// Mitsubishi GX Works2 project: KemNghiaDrillV1.5   PLC: FX3U/FX3UC

// global labels: Global1
VAR_GLOBAL
  XXLimitN AT M8344 : BOOL;
  XXLimitP AT M8343 : BOOL;
  XXBusy AT M8340 : BOOL;
  XXInterruptInverse AT M8347 : BOOL;
  XXPos AT D8340 : DINT;
  XXAccelTime AT D8348 : INT;
  XXDecelTime AT D8349 : INT;
  XXPosView AT D0 : DINT;
  XXTarPos AT D2 : DINT;
  XXFeed AT D4 : DINT;
  XXTarR AT M0 : BOOL;
  XXTarRSkip AT D6 : INT;
  XXManualN AT M1 : BOOL;
  XXManualP AT M2 : BOOL;
  XXOn AT M3 : BOOL;
  XXRun AT M4 : BOOL;
  XXDirection AT M5 : BOOL;
  XXMinI AT X000 : BOOL;
  XXAlarmI AT X004 : BOOL;
  XXReadyI AT X010 : BOOL;
  XXPulseO AT Y000 : BOOL;
  XXDirectionO AT Y004 : BOOL;
  XXOnO AT Y002 : BOOL;
  MachineReady AT M6 : BOOL;
  MachineReadyTimer AT TC0 : BOOL;
  Run AT M7 : BOOL;
  RunI AT X001 : BOOL;
  RunStop AT M8 : BOOL;
  RunStopI AT X002 : BOOL;
  RunStart AT M9 : BOOL;
  RunAuto AT M10 : BOOL;
  RunAutoEnableTimer AT TC1 : BOOL;
  RunTest AT M11 : BOOL;
  RunTestMeasureTimer AT TC246 : BOOL;
  RunTestMeasureTimerValue AT TN246 : INT;
  PositionArray AT D1000 : ARRAY [0..7] OF DINT;
  RunState AT D7 : INT;
  RunStateNext AT M12 : BOOL;
  RunStateDisc AT D8 : INT;
  RunStateDiscNext AT M13 : BOOL;
  RunStateFoilExtract AT D9 : INT;
  RunStateFoilExtractNext AT M14 : BOOL;
  RunStateDrill AT D10 : INT;
  RunStateDrillNext AT M15 : BOOL;
  RunStateFoilOut AT D11 : INT;
  RunStateFoilOutNext AT M16 : BOOL;
  DiscDRVIOffset AT D12 : DINT;
  DiscDRVIOffsetBefore AT D14 : DINT;
  DiscDRVIFrequency AT D16 : DINT;
  DiscSectorCount AT D18 : INT;
  DiscStepCount AT D19 : INT;
  DiscTest AT M17 : BOOL;
  DiscTestDelayTimer AT TC2 : BOOL;
  DiscTestMeasureTimer AT TC247 : BOOL;
  DiscTestMeasureTimerValue AT TN247 : INT;
  FoilExtractTopN AT M18 : BOOL;
  FoilExtractTopNTimer AT TC3 : BOOL;
  FoilExtractTopP AT M19 : BOOL;
  FoilExtractTopPTimer AT TC4 : BOOL;
  FoilExtractTopNI AT X003 : BOOL;
  FoilExtractTopPI AT X005 : BOOL;
  FoilExtractTop AT M20 : BOOL;
  FoilExtractTopO AT Y001 : BOOL;
  FoilExtractTopBackDelay AT D20 : INT;
  FoilExtractBotN AT M21 : BOOL;
  FoilExtractBotNTimer AT TC5 : BOOL;
  FoilExtractBotP AT M22 : BOOL;
  FoilExtractBotPTimer AT TC6 : BOOL;
  FoilExtractBotNI AT X006 : BOOL;
  FoilExtractBotPI AT X007 : BOOL;
  FoilExtractBot AT M23 : BOOL;
  FoilExtractBotO AT Y003 : BOOL;
  FoilExtractBotBackDelay AT D21 : INT;
  FoilExtractTimer AT TC7 : BOOL;
  Drill AT M24 : BOOL;
  DrillO AT Y005 : BOOL;
  DrillHold AT M25 : BOOL;
  DrillHoldO AT Y006 : BOOL;
  DrillN AT M26 : BOOL;
  DrillP AT M27 : BOOL;
  DrillNI AT X011 : BOOL;
  DrillPI AT X012 : BOOL;
  DrillIgnore AT M28 : BOOL;
  DrillIgnoreEnableTimer AT TC8 : BOOL;
  DrillIgnoreDisableTimer AT TC9 : BOOL;
  DrillIgnoreO AT Y017 : BOOL;
  DrillTimer AT TC10 : BOOL;
  FoilOutN AT M29 : BOOL;
  FoilOutNTimer AT TC11 : BOOL;
  FoilOutP AT M30 : BOOL;
  FoilOutPTimer AT TC12 : BOOL;
  FoilOutNI AT X013 : BOOL;
  FoilOutPI AT X014 : BOOL;
  FoilOut AT M31 : BOOL;
  FoilOutO AT Y007 : BOOL;
  AirBurst AT M32 : BOOL;
  AirBurstO AT Y010 : BOOL;
  AirBurstTimer AT TC13 : BOOL;
END_VAR

// task Task_01 (event TRUE, interval 0, priority 31): POU_01

PROGRAM POU_01
VAR
  fTmp : BOOL;
END_VAR
SET(M8002, M8336);
MOV(M8002, HFFF0, D8336);
RST(M8002, XXInterruptInverse);
ZRST(M8002, RunState, RunStateFoilOut);
MOV(M8002, 250, XXAccelTime);
MOV(M8002, 250, XXDecelTime);
SET(M8002, FoilExtractTop);
SET(M8002, FoilExtractBot);
RST(M8002, Drill);
MOV(M8002, 10, FoilExtractTopBackDelay);
MOV(M8002, 10, FoilExtractBotBackDelay);
RST(M8002, DiscTest);

MOV(M8002, 8, DiscSectorCount);
DMOV(M8002, 8704, XXFeed);
DMOV(M8002, 4096, PositionArray[0]);
DMOV(M8002, 4096 * 1, PositionArray[1]);
DMOV(M8002, 4096 * 2, PositionArray[2]);
DMOV(M8002, 4096 * 3, PositionArray[3]);
DMOV(M8002, 4096 * 4, PositionArray[4]);
DMOV(M8002, 4096 * 5, PositionArray[5]);
DMOV(M8002, 4096 * 6, PositionArray[6]);
DMOV(M8002, 4096 * 7, PositionArray[7]);

OUT_T(M8000 AND NOT MachineReady, MachineReadyTimer, 10);
SET(MachineReadyTimer, MachineReady);

DMOV(M8002, 128, DiscDRVIOffset);
DMOV(M8002, 256, DiscDRVIOffsetBefore); (*offset beforce must larger than offset*)
DMOV(M8002, 512, DiscDRVIFrequency);

SET(MachineReady AND Run AND RunState = 0, fTmp);
RST(fTmp, Run);
MOV(fTmp, 1, RunState);
RST(fTmp, fTmp);
SET(RunStop, fTmp);
RST(fTmp, RunStop);
ZRST(fTmp, RunState, RunStateFoilOut);
ZRST(fTmp, RunStateNext, RunStateFoilOutNext);
RST(fTmp, XXRun);
RST(fTmp, XXOn);
RST(fTmp, FoilOut);
RST(fTmp, fTmp);

INC(RunStateNext, RunState);
INC(RunStateDiscNext, RunStateDisc);
INC(RunStateFoilExtractNext, RunStateFoilExtract);
INC(RunStateDrillNext, RunStateDrill);
INC(RunStateFoilOutNext, RunStateFoilOut);
ZRST(M8000, RunStateNext, RunStateFoilOutNext);
DECO(M8000, RunState, 6, M100); 
DECO(M8000, RunStateDisc, 6, M200); DECO(M8000, RunStateDisc, 6, M1200); ZRST(NOT (XXTarR AND XXReadyI AND NOT XXAlarmI), M1200, M1263);
DECO(M8000, RunStateFoilExtract, 6, M300);
DECO(M8000, RunStateDrill, 6, M400);
DECO(M8000, RunStateFoilOut, 6, M500);

(*||||||||||Main*)
(*start run, start disc get origin*)
SET(M101, RunStart);
SET(M101, RunStateNext);
MOV(M101, 1, RunStateDisc);
(*wait disc get origin done, move to wait run command*)
MOV(M102 AND M1260, 11, RunState);
(*wait run command*)
SET(M111 AND RunAuto, fTmp);
SET(M111 AND NOT RunAuto AND Run, fTmp);
RST(fTmp, Run);
MOV(fTmp AND NOT RunStart, 21, RunStateDisc);
RST(fTmp AND RunStart, RunStart);
SET(fTmp, RunStateNext);
RST(fTmp, fTmp);
(*got run command*)
SET(M112, RunStateNext);
(*wait disc move to next position*)
SET(M113 AND M1260, RunStateNext);
(*start cycle*)
MOV(M114, 1, RunStateFoilExtract);
MOV(M114, 1, RunStateDrill);
MOV(M114, 1, RunStateFoilOut);
SET(M114, RunStateNext);
(*wait all completed, back to wait run command*)
MOV(M115 AND M1260 AND M360 AND M460 AND M560, 11, RunState);
(*test*)
RST(RunTest AND M112, RunTestMeasureTimerValue);
OUT_T(RunTest AND (M113 OR M114 OR M115), RunTestMeasureTimer, 32767);
(*||||||||||*)


(*||||||||||Disc*)
(*turn disc on*)
SET(M201 AND NOT XXOn, XXOn);
SET(M1201, RunStateDiscNext);
(*ddvi when startup*)
DDVIT(M202, PositionArray[6], 8192, XXPulseO, XXDirection);
MOV(M202 AND M8029, 11, RunStateDisc);
RST(M202 AND M8029, M202);
(*/////get origin*)
(*move fast before dvit*)
DMOVP(M1211, XXPos + PositionArray[0] - DiscDRVIOffsetBefore, XXTarPos);
SET(M1211, XXRun);
SET(M1211, RunStateDiscNext);
(*setup dvit*)
SET(M1212, RunStateDiscNext);
(*dvit*)
DDVIT(M213, DiscDRVIOffset, DiscDRVIFrequency, XXPulseO, XXDirection);
SET(M213 AND M8029, RunStateDiscNext);
RST(M213 AND M8029, M213);
(*get origin done, jump to move position done*)
RST(M1214, XXPos);
RST(M1214, DiscStepCount);
MOV(M1214, 23, RunStateDisc);
(*/////move next position*)
(*check*)
SET(M1221 AND DiscStepCount >= DiscSectorCount, fTmp);
MOV(M1221 AND fTmp, 11, RunStateDisc);
SET(M1221 AND NOT fTmp, RunStateDiscNext);
RST(fTmp, fTmp);
(*move position*)
DMOV(M1222, PositionArray[DiscStepCount], XXTarPos);
SET(M1222, XXRun);
SET(M1222, RunStateDiscNext);
(*move position done*)
INC(M1223, DiscStepCount);
MOV(M1223, 60, RunStateDisc);
(*test*)
RST(DiscTest AND M1222, DiscTestMeasureTimerValue);
OUT_T(DiscTest AND M1260, DiscTestDelayTimer, 10);
MOV(DiscTestDelayTimer, 21, RunStateDisc);
OUT_T(DiscTest AND XXRun, DiscTestMeasureTimer, 32767);
(*||||||||||*)


(*||||||||||FoilExtract*)
(*not ready, top and bot forward*)
SET(M301 AND NOT FoilExtractTopP, FoilExtractTop);
SET(M301 AND NOT FoilExtractBotP, FoilExtractBot);
RST(M301 AND NOT (FoilExtractTopP OR FoilExtractBotP), M301);
(*ready, bot back*)
RST(M301, FoilExtractBot);
SET(M301, RunStateFoilExtractNext);
(*bot back done, bot forward*)
RST(M302 AND NOT FoilExtractBotN, M302);
SET(M302, FoilExtractBot);
SET(M302, RunStateFoilExtractNext);
(*bot forward done, top back*)
OUT_T(M303, FoilExtractTimer, 5);
SET(M303 AND FoilExtractTimer AND FoilExtractBotP, fTmp);
RST(fTmp, FoilExtractTop);
SET(fTmp, RunStateFoilExtractNext);
RST(fTmp, fTmp);
(*top back done, top forward*)
RST(M304 AND NOT FoilExtractTopN, M304);
SET(M304, FoilExtractTop);
SET(M304, RunStateFoilExtractNext);
(*top forward done, end*)
MOV(M305 AND FoilExtractTopP, 60, RunStateFoilExtract);
(*||||||||||*)


(*||||||||||Drill*)
(**)
MOV(M401 AND DrillIgnore, 60, RunStateDrill);
SET(M401 AND NOT DrillIgnore, RunStateDrillNext);
(**)
SET(M402 AND DrillN, RunStateDrillNext);
(**)
SET(M403, Drill);
SET(M403, RunStateDrillNext);
(**)
SET(M404 AND NOT DrillN AND DrillP, RunStateDrillNext);
(**)
MOV(M405 AND NOT DrillP AND DrillN, 60, RunStateDrill);
(*||||||||||*)


(*||||||||||FoilOut*)
(**)
RST(M501 AND NOT FoilOutN, FoilOut);
SET(M501 AND FoilOutN, RunStateFoilOutNext);
(**)
SET(M502, FoilOut);
SET(M502, RunStateFoilOutNext);
(**)
RST(M503 AND FoilOutP, FoilOut);
SET(M503 AND FoilOutP, RunStateFoilOutNext);
(*down done, end*)
MOV(M504 AND FoilOutN, 60, RunStateFoilOut);
(*||||||||||*)

(*||||||||||*)
RST(XXRun AND XXTarPos = XXPos, XXRun);
DDRVA(XXRun, XXTarPos, XXFeed, XXPulseO, XXDirection);
RST(M8029, XXRun);
OUT(XXDirection, XXDirectionO);
INC(NOT XXRun AND NOT XXBusy AND XXTarRSkip < 5, XXTarRSkip);
RST(XXRun, XXTarRSkip);
OUT(XXTarRSkip >= 5, XXTarR);
(*||||||||||*)

(*Input*)
PLS(RunI, Run); SET(Run, Run);
PLS(RunStopI, RunStop); SET(RunStop, RunStop);
OUT_T(RunI, RunAutoEnableTimer, 20); SET(RunAutoEnableTimer, RunAuto);
OUT_T(RunStopI AND NOT DrillIgnore, DrillIgnoreEnableTimer, 20); SET(DrillIgnoreEnableTimer, DrillIgnore);
OUT_T(RunStopI AND DrillIgnore, DrillIgnoreDisableTimer, 20); RST(DrillIgnoreDisableTimer, DrillIgnore);

(**)
OUT_T(NOT FoilExtractTop, FoilExtractTopNTimer, FoilExtractTopBackDelay); SET(FoilExtractTopNTimer, FoilExtractTopN); RST(FoilExtractTopNTimer, FoilExtractTopP);
OUT_T(FoilExtractTopPI, FoilExtractTopPTimer, 3); SET(FoilExtractTopPTimer, FoilExtractTopP); RST(FoilExtractTopPTimer, FoilExtractTopN);
(**)
OUT_T(NOT FoilExtractBot, FoilExtractBotNTimer, FoilExtractBotBackDelay); SET(FoilExtractBotNTimer, FoilExtractBotN); RST(FoilExtractBotNTimer, FoilExtractBotP);
OUT_T(FoilExtractBotPI, FoilExtractBotPTimer, 3); SET(FoilExtractBotPTimer, FoilExtractBotP); RST(FoilExtractBotPTimer, FoilExtractBotN);
(**)

(**)
OUT_T(FoilOutNI, FoilOutNTimer, 3); SET(FoilOutNTimer, FoilOutN); RST(FoilOutNTimer, FoilOutP);
OUT_T(FoilOutPI, FoilOutPTimer, 3); SET(FoilOutPTimer, FoilOutP); RST(FoilOutPTimer, FoilOutN);
(**)

(*Output*)
OUT_T(AirBurst, AirBurstTimer, 10); RST(AirBurstTimer, AirBurst);
OUT_T(Drill, DrillTimer, 2); RST(DrillTimer, Drill);
(**)
OUT(XXOn, XXOnO);
OUT(NOT FoilExtractTop, FoilExtractTopO);
OUT(NOT FoilExtractBot, FoilExtractBotO);
OUT(Drill, DrillO);
OUT(DrillIgnore, DrillIgnoreO);
OUT(FoilOut, FoilOutO);
OUT(AirBurst, AirBurstO);
END_PROGRAM
